PROGRAM PRG_LOG
VAR
    fbLogHandler: FB_LogHandler;
END_VAR

fbLogHandler();

END_PROGRAM

(* stored: Version 1.1.0.1
   POU PRG_LOG: Id {a40ec52b-fefa-047d-21a6-a40c23d32a5a}, SpecialFunc None *)
